// TIA Portal V17 export
// export: Created 2025-06-26T07:49:42.8141093Z, ExportSetting WithDefaults, DisplayName Totally Integrated Automation Portal, DisplayVersion V17 Update 8, DisplayName TIA Portal Openness, DisplayVersion V17 Update 8, DisplayName TIA Portal Version Control Interface, DisplayVersion V17, DisplayName STEP 7 Professional, DisplayVersion V17 Update 8, DisplayName STEP 7 Safety, DisplayVersion V17 Update 6, DisplayName WinCC Advanced, DisplayVersion V17 Update 8
DATA_BLOCK "Diagnosis_DB"   // DB1
VERSION : 0.1
// stored: AutoNumber true, DBAccessibleFromOPCUA true, DBAccessibleFromWebserver true, InstanceOfName Diagnosis, InstanceOfType FB
"Diagnosis"
   // VAR
   //    A0001 { ExternalAccessible := 'False'; ExternalVisible := 'False'; ExternalWritable := 'False'} : "fbHMIEvent";
   //    A1002 { ExternalAccessible := 'False'; ExternalVisible := 'False'; ExternalWritable := 'False'; S7_SetPoint := 'True'} : "fbHMIEvent";
   //    A1003 { ExternalAccessible := 'False'; ExternalVisible := 'False'; ExternalWritable := 'False'; S7_SetPoint := 'True'} : "fbHMIEvent";
   // END_VAR
BEGIN
END_DATA_BLOCK
